// TIA Portal V17 export
// export: Created 2024-08-07T21:44:11.8858435Z, ExportSetting WithDefaults, DisplayName Totally Integrated Automation Portal, DisplayVersion V17 Update 7, DisplayName TIA Portal Openness, DisplayVersion V17 Update 7, DisplayName TIA Portal Version Control Interface, DisplayVersion V17, DisplayName SINAMICS Startdrive Advanced, DisplayVersion V17 SP2, DisplayName SINAMICS Startdrive G110M, G120, G120C, G120D, G120P, G115D, DisplayVersion V17 SP2, DisplayName SINAMICS Startdrive G130, G150, S120, S150, SINAMICS MV, S210, DisplayVersion V17 SP2, DisplayName STEP 7 Professional, DisplayVersion V17 Update 7, DisplayName STEP 7 Safety, DisplayVersion V17 Update 6, DisplayName WinCC Advanced / Unified PC, DisplayVersion V17 Update 7
DATA_BLOCK "MII_Parameters"   // DB2020
{ S7_Optimized_Access := 'TRUE' }
VERSION : 0.1
// stored: AutoNumber false, DBAccessibleFromOPCUA true, DBAccessibleFromWebserver true, IsOnlyStoredInLoadMemory false, IsRetainMemResEnabled false, IsWriteProtectedInAS false, MemoryReserve 100
   VAR RETAIN
      Connection : Struct
         IPAddress : WString := WSTRING#'10.223.41.34';   // Server IP Address (e.g. 10.223.41.34)
         ServerPort : WString := WSTRING#'58710/PCoUaServer';   // Server port (e.g. 58710)
         PlantID : WString := WSTRING#'P2';   // Unique plant id defined by local DMC key user (e.g. P1 or P2)
         PLC_ID : WString := WSTRING#'1300T1';   // Unique plc id defined by local DMC key user (different from ijcore)
         OperationMode : Bool;   // False: production; True: test
      END_STRUCT;
   END_VAR
   VAR
      Commands : Struct
         getLocalTime : Bool;   // Forces the call for local time
         testProdDeclaration : Bool;   // Forces the call for production declaration
         auxTestProdDeclaration : Int := 1;   // Auxiliar counter for testing
         forceReconnection : Bool;   // Forces the reconnection to the server
      END_STRUCT;
   END_VAR
   VAR RETAIN
      Connection_Status : Struct
         opcUaConnected : Bool;   // True if the client if connected to the server
         opcUaError : Bool;   // True if error during connection attempt
         opcUaStatus : Word;
         opcUaDiagnostics : DWord;   // Detailed error information
         aux : Struct
            diagnosticStatus : DInt;
            opcUaSubfunctionStatus : DInt;
            nAttemptsTotal : Int := 1;
         END_STRUCT;
      END_STRUCT;
      M000_Status : Struct
         error : Bool;   // True if an error occurred during method call
         status : WString;   // Detailed error information
         timestamp : LDT;   // Timestamp of method call attempt
         Inputs : "MII_Interface.MII_METHODS.M000_PRODUCTION_DECLARATION.Inputs";   // Input arguments during error
         Outputs { S7_SetPoint := 'True'} : "MII_Interface.MII_METHODS.M000_PRODUCTION_DECLARATION.Outputs";   // Output arguments during error
      END_STRUCT;
      M002_Status : Struct
         localTime : LDT;   // Last system time received
         status : WString;   // Status of method call
      END_STRUCT;
   END_VAR
   VAR
      HMI : Struct
         statusHmiDMC1 : Int;
         statusHmiDMC2 : Int;
      END_STRUCT;
   END_VAR
   VAR RETAIN
      optionSt1St2 : Bool;   // option for C2P if it's ON product declaration split for ST1/ST2
   END_VAR
BEGIN
END_DATA_BLOCK
